(* IEC 61131-3 sources: model/new_model/baseline/data/sample, 6 files *)

(* ---- arr_oob_1.st ---- *)
PROGRAM arr_oob_1
VAR
  buf : ARRAY[0..9] OF INT;
  i : INT;
END_VAR
buf[i + 1] := 5;
END_PROGRAM

(* ---- arr_oob_2.st ---- *)
PROGRAM arr_oob_2
VAR
  tank_levels : ARRAY[0..3] OF REAL;
  idx : INT;
END_VAR
tank_levels[idx + 2] := 99.0;
END_PROGRAM

(* ---- clean_1.st ---- *)
PROGRAM clean_1
VAR
  a : INT := 0;
  b : INT := 1;
END_VAR
a := b + 2;
END_PROGRAM

(* ---- clean_2.st ---- *)
PROGRAM clean_2
VAR
  motor_speed : INT := 0;
  setpoint : INT := 50;
END_VAR
motor_speed := setpoint - 5;
END_PROGRAM

(* ---- div_zero_1.st ---- *)
PROGRAM div_zero_1
VAR
  x : INT;
  y : INT;
END_VAR
y := x / 0;
END_PROGRAM

(* ---- div_zero_2.st ---- *)
PROGRAM div_zero_2
VAR
  flow : REAL;
  rate : REAL;
END_VAR
rate := flow / 0;
END_PROGRAM
